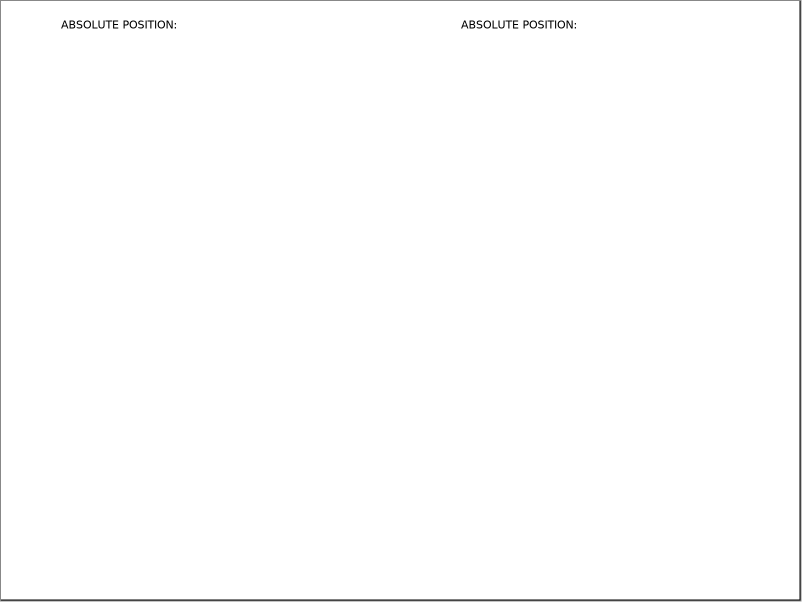
VISUALIZATION F14_Read_Actual_Torque  // 802x602
    Rectangle (0,0 800x600)
    Label (10,10 170x30), "ABSOLUTE POSITION:"
    Label (410,10 170x30), "ABSOLUTE POSITION:"
END_VISUALIZATION

(* stored: Version 1.1.0.1, ProductVersion 3.1.4022.7
   Visu F14_Read_Actual_Torque: Id {afa8c62b-8314-4920-947f-9d491e690ba2} *)
